PROGRAM MAIN
VAR
END_VAR

END_PROGRAM

(* stored: Version 1.1.0.1
   POU MAIN: Id {183ba2ae-5ddc-4dea-9599-53c21335e6f8} *)
